PROGRAM PRG_Simulation
VAR
	fAxis3SimulationActPosY: LREAL;
	bParca1Invisible: BOOL;
	bParca2Invisible2: BOOL;
	fAxis1SimulationActPosX: LREAL;

	fAxis2SimulationActPosX: LREAL;
	bMatkapInvisible: BOOL;
	bMatkapInvisible2: BOOL;
	bMatkapInvisible3: BOOL;
	nState: INT;
	nUp: INT;
	bParcaUpInvisible: BOOL;
	nRight: INT;
	bParcaRightInvisible: BOOL;
	t1: TON;
	bAxis31000Position: BOOL;
END_VAR

IF Axis1.NcToPlc.ActPos >= 6000 AND Axis1.NcToPlc.ActPos < 20000 THEN
	bParca1Invisible		:= TRUE;
	bParca2Invisible2		:= FALSE;
	fAxis1SimulationActPosX	:= (Axis1.NcToPlc.ActPos-6000)/30;
ELSIF Axis1.NcToPlc.ActPos >= 20000 THEN
	bParca2Invisible2		:= TRUE;
	bAxis31000Position		:= FALSE;
	fAxis3SimulationActPosY	:= 0;
ELSIF Axis1.NcToPlc.ActPos=0 OR Axis1.NcToPlc.ActPos<1 THEN
	bParca2Invisible2		:= TRUE;
END_IF

IF Axis2.NcToPlc.ActPos>=1000 AND Axis2.Status.PositiveDirection THEN
	fAxis2SimulationActPosX	:= (Axis2.NcToPlc.ActPos-1000)/30;
	bMatkapInvisible		:= TRUE;
	bMatkapInvisible2		:= FALSE;
ELSIF Axis2.NcToPlc.ActPos=0 OR Axis2.NcToPlc.ActPos<1 THEN
	bMatkapInvisible		:= FALSE;
	bMatkapInvisible3		:= TRUE;
	bMatkapInvisible2		:= TRUE;
END_IF


IF Axis2.Status.NegativeDirection THEN
	fAxis2SimulationActPosX	:= (Axis2.NcToPlc.ActPos)/30;
	bMatkapInvisible	:= TRUE;
	bMatkapInvisible2	:= TRUE;
	bMatkapInvisible3	:= FALSE;
END_IF

IF Axis3.NcToPlc.ActPos>=692.3076921 AND NOT bAxis31000Position THEN
	fAxis3SimulationActPosY	:= (Axis3.NcToPlc.ActPos/15.38461538)-45;
END_IF

IF  Axis3.NcToPlc.ActPos>=999 THEN
	fAxis3SimulationActPosY	:= 20;
	bAxis31000Position		:= TRUE;
END_IF

CASE nState OF

0:
	.bStartSensor	:= FALSE;
	IF NOT .bProcessActive THEN
		.bEnable	:= TRUE;
		nState		:= 10;
		bParcaUpInvisible	:= FALSE; 
	END_IF

10:
	nUp						:= nUp+1;
	IF nUp>=135 THEN
		nState				:= 20;
	END_IF
	
20:
	nRight					:= nRight+1;
	IF nRight>=61 THEN
		bParcaUpInvisible	:= TRUE; 
		nState				:= 25;
		bParca1Invisible		:= FALSE;
	END_IF
	
25:
	nRight					:= nRight-1;
	IF nRight<=0 THEN		
		nState				:= 27;	
	END_IF

27:
	nUp						:= nUp-1;
	IF nUp<=0 THEN
		nState				:= 30;
	END_IF
30:
	bStartSensor				:= TRUE;
	t1(IN:= TRUE , PT:= T#30MS , Q=> , ET=> );
	IF t1.Q THEN
		t1(IN:= FALSE);
		nState						:= 0;
		nRight						:= 0;
		nUp							:= 0;
	END_IF

END_CASE

END_PROGRAM

(* stored: Version 1.1.0.1, ProductVersion 3.1.4022.12
   POU PRG_Simulation: Id {49b9eab7-c0f0-4232-bb02-e8fa5328da03}, SpecialFunc None *)
